TYPE ST_MyStruct :
STRUCT
	A, B, C : INT;
	Value : REAL;
	Descr : STRING;
END_STRUCT
END_TYPE

(* stored: Version 1.1.0.1, ProductVersion 3.1.4024.4
   DUT ST_MyStruct: Id {d6e56e52-60aa-4123-81f6-6771d7bc6a67} *)
